PROGRAM PRG_SFLX_01_TransportConvCtrl
VAR
	fbPerformance				: FB_Interval;

	tofTransferConvDelay		: FB_TOFR;
	rsOuterAtTransferStation	: RS;
	tonTransferTimeout		: TON;
END_VAR

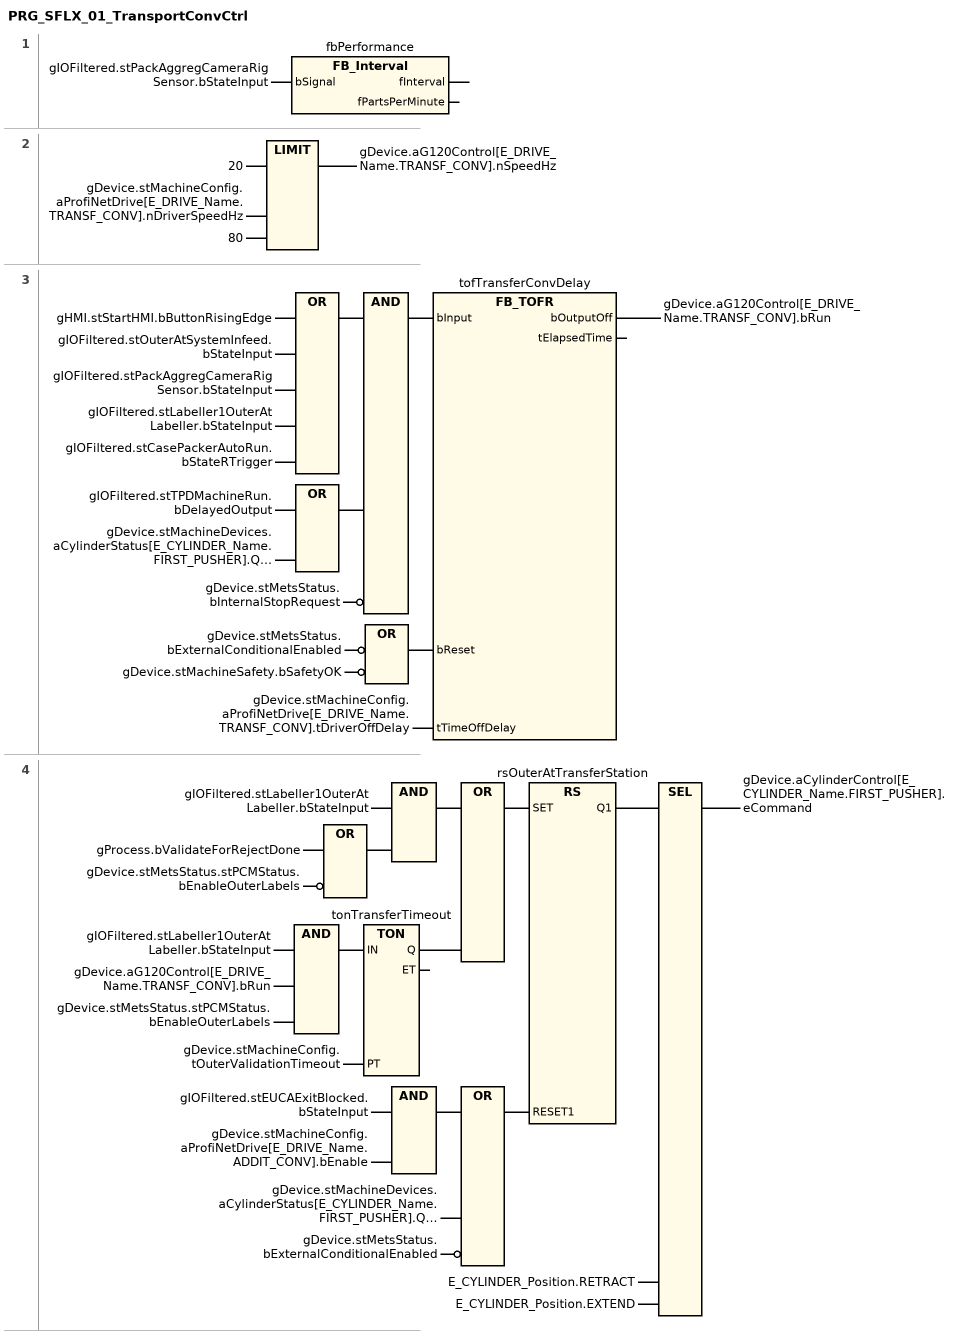
// NETWORK 1
fbPerformance(bSignal := gIOFiltered.stPackAggregCameraRigSensor.bStateInput); // FB_Interval

// NETWORK 2
gDevice.aG120Control[E_DRIVE_Name.TRANSF_CONV].nSpeedHz := LIMIT(20, gDevice.stMachineConfig.aProfiNetDrive[E_DRIVE_Name.TRANSF_CONV].nDriverSpeedHz, 80);

// NETWORK 3
tofTransferConvDelay(
    bInput := (gHMI.stStartHMI.bButtonRisingEdge OR gIOFiltered.stOuterAtSystemInfeed.bStateInput OR gIOFiltered.stPackAggregCameraRigSensor.bStateInput OR gIOFiltered.stLabeller1OuterAtLabeller.bStateInput OR gIOFiltered.stCasePackerAutoRun.bStateRTrigger) AND (gIOFiltered.stTPDMachineRun.bDelayedOutput OR gDevice.stMachineDevices.aCylinderStatus[E_CYLINDER_Name.FIRST_PUSHER].Q.bCylinderInExtendedPosition) AND NOT gDevice.stMetsStatus.bInternalStopRequest,
    bReset := NOT gDevice.stMetsStatus.bExternalConditionalEnabled OR NOT gDevice.stMachineSafety.bSafetyOK,
    tTimeOffDelay := gDevice.stMachineConfig.aProfiNetDrive[E_DRIVE_Name.TRANSF_CONV].tDriverOffDelay); // FB_TOFR
gDevice.aG120Control[E_DRIVE_Name.TRANSF_CONV].bRun := tofTransferConvDelay.bOutputOff;

// NETWORK 4
tonTransferTimeout(IN := gIOFiltered.stLabeller1OuterAtLabeller.bStateInput AND gDevice.aG120Control[E_DRIVE_Name.TRANSF_CONV].bRun AND gDevice.stMetsStatus.stPCMStatus.bEnableOuterLabels, PT := gDevice.stMachineConfig.tOuterValidationTimeout); // TON
rsOuterAtTransferStation(SET := gIOFiltered.stLabeller1OuterAtLabeller.bStateInput AND (gProcess.bValidateForRejectDone OR NOT gDevice.stMetsStatus.stPCMStatus.bEnableOuterLabels) OR tonTransferTimeout.Q, RESET1 := gIOFiltered.stEUCAExitBlocked.bStateInput AND gDevice.stMachineConfig.aProfiNetDrive[E_DRIVE_Name.ADDIT_CONV].bEnable OR gDevice.stMachineDevices.aCylinderStatus[E_CYLINDER_Name.FIRST_PUSHER].Q.bCylinderInExtendedPosition OR NOT gDevice.stMetsStatus.bExternalConditionalEnabled); // RS
gDevice.aCylinderControl[E_CYLINDER_Name.FIRST_PUSHER].eCommand := SEL(rsOuterAtTransferStation.Q1, E_CYLINDER_Position.RETRACT, E_CYLINDER_Position.EXTEND);

END_PROGRAM

(* stored: Version 1.1.0.1
   POU PRG_SFLX_01_TransportConvCtrl: Id {251831c0-759c-4081-817c-4136524beb00}, SpecialFunc None *)
